(*

.. <legal notes>

legal notes
=================
| SPDX-FileCopyrightText: © 2026 Oleksandr Tiutyk <trofimich@gmail.com>
| SPDX-License-Identifier: LGPL-3.0-only
| For details check: LGPL-3.0-only_

.. _LGPL-3.0-only: https://www.gnu.org/licenses/lgpl-3.0.en.html

.. </legal notes>

*)

PROGRAM UsignedByteHelper
VAR CONSTANT
	MIN_VALUE : BYTE := 0;
	MAX_VALUE : BYTE := 255;
END_VAR
VAR
	_ClassName : STRING := __POUNAME();
END_VAR

{attribute 'monitoring' := 'call'}
PROPERTY ClassName : STRING
GET
ClassName := _ClassName;
END_GET
END_PROPERTY

{attribute 'monitoring' := 'call'}
PROPERTY NamespaceName : STRING
GET
NamespaceName := CurrentNamespace.Name;
END_GET
END_PROPERTY

END_PROGRAM

(* stored: Version 1.1.0.1
   POU UsignedByteHelper: Id {4535912c-7c28-45af-ab90-74f12bea42b1}, SpecialFunc None
   Property ClassName: Id {7cdfd4b8-4143-436d-8a80-d8d11af812c3}
   Get Get: Id {a66bdd50-80ee-42c4-8efa-220958ec5c8a}
   Property NamespaceName: Id {7eb551b0-be22-4fd0-8050-6706a2730601}
   Get Get: Id {53ee3327-4ef7-469b-8356-c1c023ceb189} *)
